FUNCTION ST08B_TO_BOOLS
  (* Standard: 61499-1; Description: Copyright (c) 2024 HR Agrartechnik GmbH This program and the accompanying materials are made available under the terms of the Eclipse Public License 2.0 which is available at https://www.eclipse.org/legal/epl-2.0/ SPDX-License-Identifier: EPL-2.0 *)
  (* Version 1.0, 2024-02-22, Franz Höpfinger, HR Agrartechnik GmbH *)
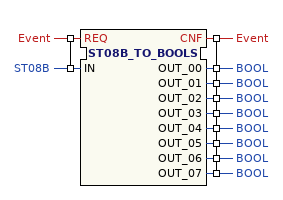
  EVENT_INPUT
    REQ WITH IN; (* Normal Execution Request *)
  END_EVENT
  EVENT_OUTPUT
    CNF WITH OUT_00, OUT_01, OUT_02, OUT_03, OUT_04, OUT_05, OUT_06, OUT_07; (* Execution Confirmation *)
  END_EVENT
  VAR_INPUT
    IN : ST08B; (* ST08B Input *)
  END_VAR
  VAR_OUTPUT
    OUT_00 : BOOL; (* BIT 00 *)
    OUT_01 : BOOL; (* BIT 01 *)
    OUT_02 : BOOL; (* BIT 02 *)
    OUT_03 : BOOL; (* BIT 03 *)
    OUT_04 : BOOL; (* BIT 04 *)
    OUT_05 : BOOL; (* BIT 05 *)
    OUT_06 : BOOL; (* BIT 06 *)
    OUT_07 : BOOL; (* BIT 07 *)
  END_VAR
  BODY IN ST:
FUNCTION ST08B_TO_BOOLS

VAR_INPUT
	IN : ST08B;    // ST08B Input
END_VAR

VAR_OUTPUT
	OUT_00 : BOOL;    // BIT 00
	OUT_01 : BOOL;    // BIT 01
	OUT_02 : BOOL;    // BIT 02
	OUT_03 : BOOL;    // BIT 03
	OUT_04 : BOOL;    // BIT 04
	OUT_05 : BOOL;    // BIT 05
	OUT_06 : BOOL;    // BIT 06
	OUT_07 : BOOL;    // BIT 07
END_VAR

(* this Function extracts the 8 BOOLS from a byte *)
OUT_00 := IN.B_00;
OUT_01 := IN.B_01;
OUT_02 := IN.B_02;
OUT_03 := IN.B_03;
OUT_04 := IN.B_04;
OUT_05 := IN.B_05;
OUT_06 := IN.B_06;
OUT_07 := IN.B_07;

END_FUNCTION
  END_BODY
END_FUNCTION
